(* Logix 5000 project; controller GEA_Test_Chamber vendor 1 type 14 code 196 rev 32.14; software revision 32.04; part 2 of 11 *)
(* tags used below, declared in another part *)
   Ref_Transactions : raC_UDT_ModbusClientTransaction[5];
   Sts_Overlap : BOOL;
   Sts_Overload : BOOL;
   Wrk_Main_Read_Buffer : STR4096;
   Wrk_ArraySize : DINT;
   Wrk_LastTransaction : DINT;
   Wrk_tempHMItransaction : DINT;
   Wrk_HMITransactionValid : BOOL;
(* raC_Opr_NetModbusTCPClient, continued *)

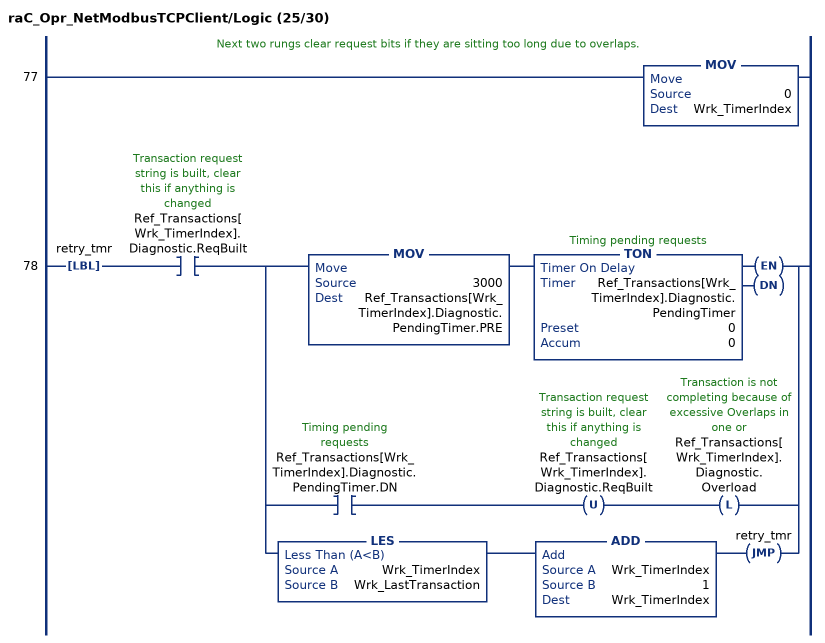
   // Next two rungs clear request bits if they are sitting too long due to overlaps.
   77: MOV(0,Wrk_TimerIndex);
   78: LBL(retry_tmr)XIC(Ref_Transactions[Wrk_TimerIndex].Diagnostic.ReqBuilt)[MOV(3000,Ref_Transactions[Wrk_TimerIndex].Diagnostic.PendingTimer.PRE) TON(Ref_Transactions[Wrk_TimerIndex].Diagnostic.PendingTimer,0,0) ,XIC(Ref_Transactions[Wrk_TimerIndex].Diagnostic.PendingTimer.DN) OTU(Ref_Transactions[Wrk_TimerIndex].Diagnostic.ReqBuilt) OTL(Ref_Transactions[Wrk_TimerIndex].Diagnostic.Overload) ,LES(Wrk_TimerIndex,Wrk_LastTransaction) ADD(Wrk_TimerIndex,1,Wrk_TimerIndex) JMP(retry_tmr) ];
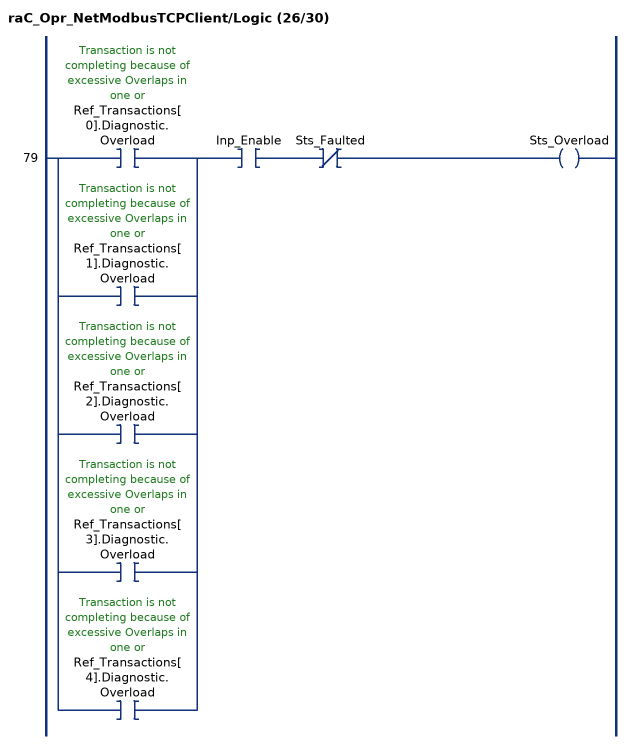
   79: [XIC(Ref_Transactions[0].Diagnostic.Overload) ,XIC(Ref_Transactions[1].Diagnostic.Overload) ,XIC(Ref_Transactions[2].Diagnostic.Overload) ,XIC(Ref_Transactions[3].Diagnostic.Overload) ,XIC(Ref_Transactions[4].Diagnostic.Overload) ]XIC(Inp_Enable)XIO(Sts_Faulted)OTE(Sts_Overload);
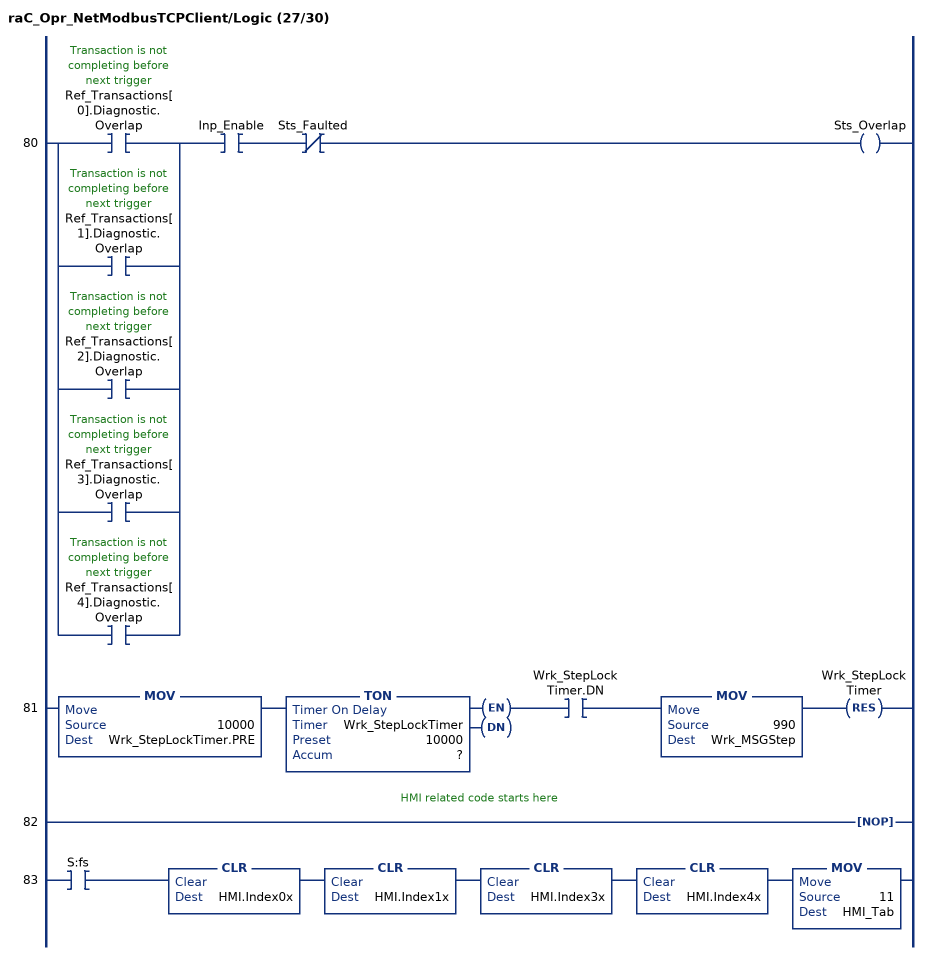
   80: [XIC(Ref_Transactions[0].Diagnostic.Overlap) ,XIC(Ref_Transactions[1].Diagnostic.Overlap) ,XIC(Ref_Transactions[2].Diagnostic.Overlap) ,XIC(Ref_Transactions[3].Diagnostic.Overlap) ,XIC(Ref_Transactions[4].Diagnostic.Overlap) ]XIC(Inp_Enable)XIO(Sts_Faulted)OTE(Sts_Overlap);
   81: MOV(10000,Wrk_StepLockTimer.PRE)TON(Wrk_StepLockTimer,?,?)XIC(Wrk_StepLockTimer.DN)MOV(990,Wrk_MSGStep)RES(Wrk_StepLockTimer);
   // HMI related code starts here
   82: NOP();
   83: XIC(S:fs)CLR(HMI.Index0x)CLR(HMI.Index1x)CLR(HMI.Index3x)CLR(HMI.Index4x)MOV(11,HMI_Tab);
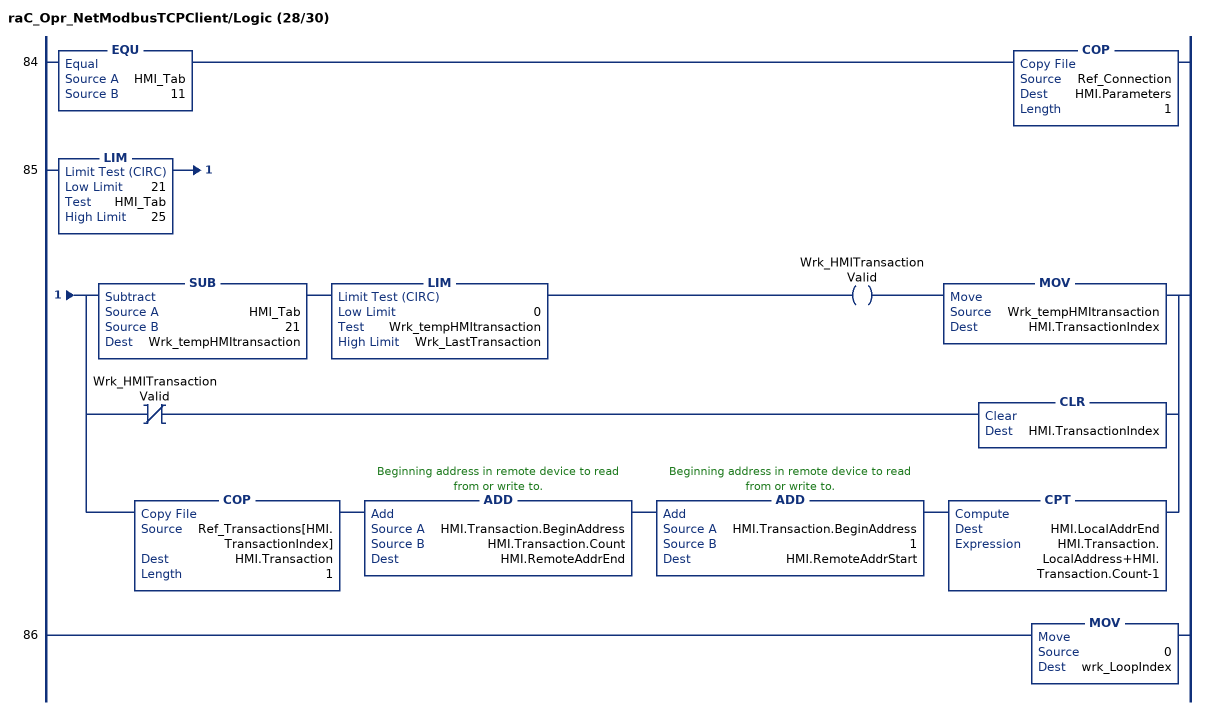
   84: EQU(HMI_Tab,11)COP(Ref_Connection,HMI.Parameters,1);
   85: LIM(21,HMI_Tab,25)[SUB(HMI_Tab,21,Wrk_tempHMItransaction) LIM(0,Wrk_tempHMItransaction,Wrk_LastTransaction) OTE(Wrk_HMITransactionValid) MOV(Wrk_tempHMItransaction,HMI.TransactionIndex) ,XIO(Wrk_HMITransactionValid) CLR(HMI.TransactionIndex) ,COP(Ref_Transactions[HMI.TransactionIndex],HMI.Transaction,1) ADD(HMI.Transaction.BeginAddress,HMI.Transaction.Count,HMI.RemoteAddrEnd) ADD(HMI.Transaction.BeginAddress,1,HMI.RemoteAddrStart) CPT(HMI.LocalAddrEnd,HMI.Transaction.LocalAddress+HMI.Transaction.Count-1) ];
   86: MOV(0,wrk_LoopIndex);
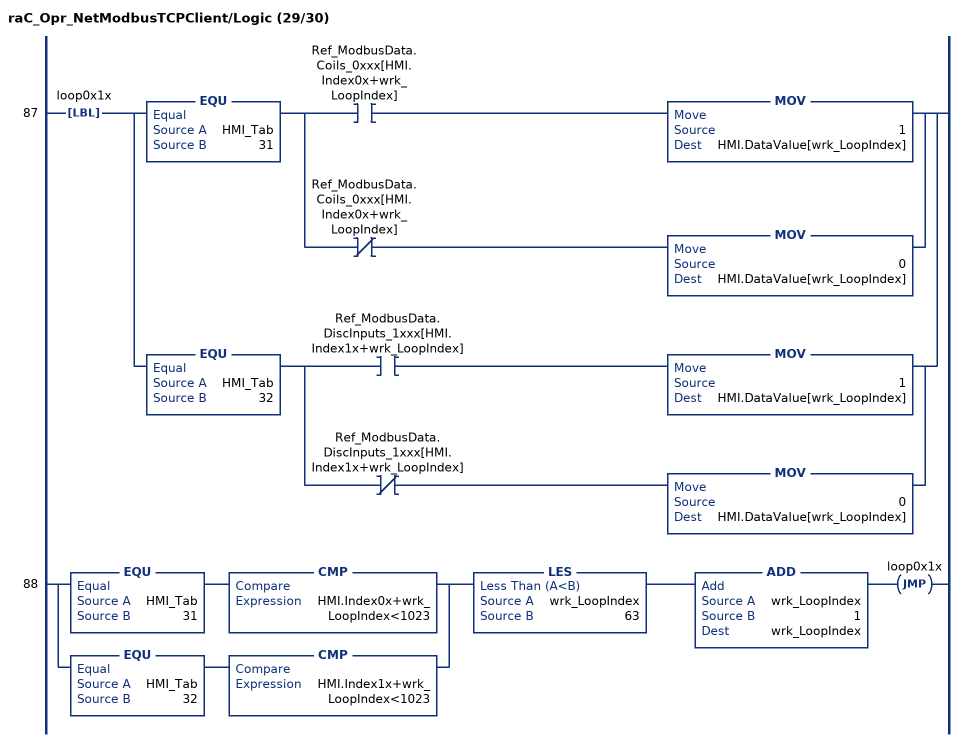
   87: LBL(loop0x1x)[EQU(HMI_Tab,31) [XIC(Ref_ModbusData.Coils_0xxx[HMI.Index0x+wrk_LoopIndex]) MOV(1,HMI.DataValue[wrk_LoopIndex]) ,XIO(Ref_ModbusData.Coils_0xxx[HMI.Index0x+wrk_LoopIndex]) MOV(0,HMI.DataValue[wrk_LoopIndex]) ] ,EQU(HMI_Tab,32) [XIC(Ref_ModbusData.DiscInputs_1xxx[HMI.Index1x+wrk_LoopIndex]) MOV(1,HMI.DataValue[wrk_LoopIndex]) ,XIO(Ref_ModbusData.DiscInputs_1xxx[HMI.Index1x+wrk_LoopIndex]) MOV(0,HMI.DataValue[wrk_LoopIndex]) ] ];
   88: [EQU(HMI_Tab,31) CMP(HMI.Index0x+wrk_LoopIndex<1023) ,EQU(HMI_Tab,32) CMP(HMI.Index1x+wrk_LoopIndex<1023) ]LES(wrk_LoopIndex,63)ADD(wrk_LoopIndex,1,wrk_LoopIndex)JMP(loop0x1x);
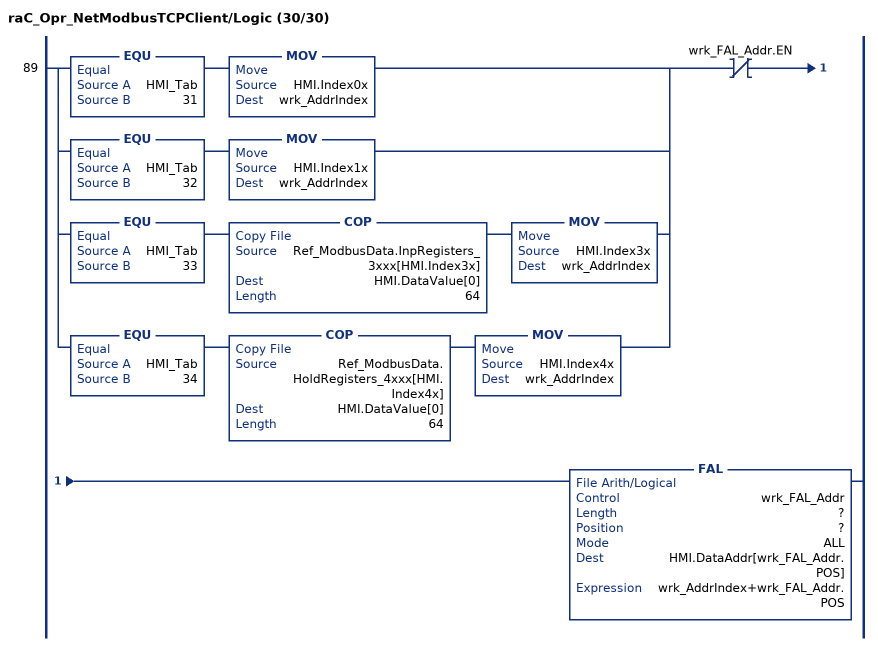
   89: [EQU(HMI_Tab,31) MOV(HMI.Index0x,wrk_AddrIndex) ,EQU(HMI_Tab,32) MOV(HMI.Index1x,wrk_AddrIndex) ,EQU(HMI_Tab,33) COP(Ref_ModbusData.InpRegisters_3xxx[HMI.Index3x],HMI.DataValue[0],64) MOV(HMI.Index3x,wrk_AddrIndex) ,EQU(HMI_Tab,34) COP(Ref_ModbusData.HoldRegisters_4xxx[HMI.Index4x],HMI.DataValue[0],64) MOV(HMI.Index4x,wrk_AddrIndex) ]XIO(wrk_FAL_Addr.EN)FAL(wrk_FAL_Addr,?,?,ALL,HMI.DataAddr[wrk_FAL_Addr.POS],wrk_AddrIndex+wrk_FAL_Addr.POS);
END_ROUTINE

ROUTINE Prescan   (* ladder *)
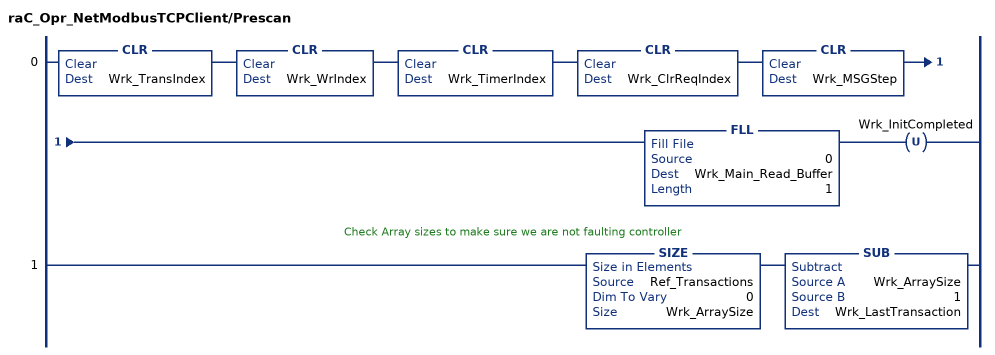
   0: CLR(Wrk_TransIndex)CLR(Wrk_WrIndex)CLR(Wrk_TimerIndex)CLR(Wrk_ClrReqIndex)CLR(Wrk_MSGStep)FLL(0,Wrk_Main_Read_Buffer,1)OTU(Wrk_InitCompleted);
   // Check Array sizes to make sure we are not faulting controller
   1: SIZE(Ref_Transactions,0,Wrk_ArraySize)SUB(Wrk_ArraySize,1,Wrk_LastTransaction);
END_ROUTINE
END_ADD_ON_INSTRUCTION

ADD_ON_INSTRUCTION raC_Opr_NetModbusTCPServer   (* revision 2.3 0, vendor Rockwell Automation, ExecutePrescan *)
// Modbus TCP Server
// Revision note:
// 2.0.0 Initial release in AOI format
// 2.0.1 Corrected local IP address logic
// 2.1.0 Corrected power-up and Redundancy anomalies
// 2.2.0 Force LocalSlot 0 for CompactLogix
// 2.3.0 Added incoming Client IP address reference tag and HMI structure
VAR_INPUT
   Inp_Enable : BOOL; {required}
END_VAR
VAR_IN_OUT
   Ref_Connection : raC_UDT_ModbusServerBase; {required}
   Ref_ModbusData : raC_UDT_ModbusServerData; {required}
END_VAR
VAR_OUTPUT
   Sts_ActiveConnections : DINT; {access Read Only, visible}   // Number of currently active Client connections.
END_VAR
VAR_IN_OUT
   Ref_MsgCreate : MESSAGE; {required}
   Ref_MsgAccept : MESSAGE; {required}
   Ref_MsgRead : MESSAGE; {required}
   Ref_MsgWrite : MESSAGE; {required}
   Ref_MsgDelete : MESSAGE; {required}
   Ref_MsgDeleteAll : MESSAGE; {required}
   Ref_MsgSetAttrSingle : MESSAGE; {required}
END_VAR
VAR_OUTPUT
   Sts_EN : BOOL; {access Read Only, visible}
   Sts_Waiting : BOOL; {access Read Only, visible}
   Sts_Accepted : BOOL; {access Read Only, visible}
   Sts_Faulted : BOOL; {access Read Only, visible}
   Sts_LastError : DINT; {access Read Only}   // The last recorded socket error for this connection. 0 good, -2- Write Error, -4 - Read Error, -6 connection failed, -7 Delete all failed, -8 Create Soc failed, -9 Connection failed, -10 connection dropped, -11 error in setting socket parameter. -12 - Enable removed -15 - Max number of connected clients exceeded
END_VAR
VAR
   Wrk_MSGStep : DINT; {access None}
   Wrk_CreateReq : raC_UDT_ModbusCreateParam; {access None}
   Wrk_BaseInstance : DINT; {access None}
   Wrk_NoreplyCounter : DINT; {access None}
   Wrk_RetryTimer : TIMER := (PRE := 5000); {access None}
   Wrk_MSGRead_SRC : DINT[2]; {access None}   // User for MSG Read Source
   Wrk_TempString : STR0462; {access None}
   Wrk_WrIndex : DINT; {access None}
   Wrk_TempDINT : DINT; {access None}
   Wrk_AdditionalLen : INT; {access None}
   Wrk_AdditionaLenRead : INT; {access None}
   Wrk_ModbusCmdLen : INT; {access None}
   Wrk_AdditionalLen1 : INT; {access None}
   Wrk_ModbusPacket : STR0462; {access None}
   Wrk_DataReceived : BOOL; {access None}
   Wrk_CmdFromReadPacket : DINT; {access None}
   Wrk_ModbusID : STR0008; {access None}
   Wrk_TempInt : INT; {access None}
   Wrk_ModbusCmdStart : INT; {access None}
   Wrk_ModbusUnit : STR0008; {access None}
   Wrk_ModbusBytes : DINT; {access None}
   Wrk_ModbusCmdString : STR0462; {access None}
   Wrk_RSB : raC_Tec_NetModbusTCPServer_RespStrBit; {access None}
   Wrk_TransIndex : DINT; {access None}
   Wrk_TimerIndex : DINT; {access None}
   Wrk_RSW : raC_Tec_NetModbusTCPServer_RespStrWord; {access None}
   Wrk_TempOctet : DINT[4]; {access None}
   Wrk_TempStrOctet : STR0008; {access None}
   Wrk_TempStrOctetlen : DINT; {access None}
   Wrk_TempIPStr : STR0016; {access None}
   Wrk_ClrReqIndex : DINT; {access None}
   Wrk_ListenSocketLost : BOOL; {access None}
   Wrk_AcceptInstance : DINT; {access None}
   Wrk_FES : raC_Tec_NetModbusTCPServer_FndEmptySckt; {access None}
   Wrk_InstSize : DINT; {access None}
   Wrk_RdWrIndex : DINT; {access None}
   Wrk_ModbusRespString : STR0462; {access None}
   Wrk_TempActConn : DINT; {access None}
   Wrk_InstIndex : DINT; {access None}
   Wrk_LastInstIndex : DINT; {access None}
   Wrk_OkToIncement : BOOL; {access None}
   Wrk_CmdFromReadPacketTmp : DINT; {access None}
   Wrk_StepLockTimer : TIMER := (PRE := 10000); {access None}
   Wrk_TempTime : DINT; {access None}
   Wrk_OktoCheckAccept : BOOL; {access None}
   Wrk_OkToIncement320 : BOOL; {access None}
   Wrk_Instances : raC_UDT_ModbusServerRWSocket[10]; {access Read Only}
   Wrk_Controller_Type : DINT; {access None}
   Wrk_Controller_Name : SINT[33]; {access None}
   Wrk_InitCompleted : BOOL; {access None}
   Wrk_AcceptAddress : DINT; {access None}
   Wrk_InstIndex2 : DINT; {access None}
   Wrk_InstIndex3 : DINT; {access None}
   HMI_Tab : DINT;
   Inf_Lib : STR0016; {access Read Only}
   Inf_Type : STR0032; {access Read Only}
   Inf_Version : STR0016; {access Read Only}
   wrk_temp_Instances : raC_UDT_ModbusServerRWSocketInfo[10]; {access None}
   wrk_FAL_Addr : CONTROL := (LEN := 64); {access None}
   wrk_LoopIndex : DINT; {access None}
   wrk_AddrIndex : DINT; {access None}
   HMI : raC_UDT_ModbusServerHMI;
   wrk_FAL_01 : CONTROL := (LEN := 10); {access None}
END_VAR

ROUTINE Logic   (* ladder *)
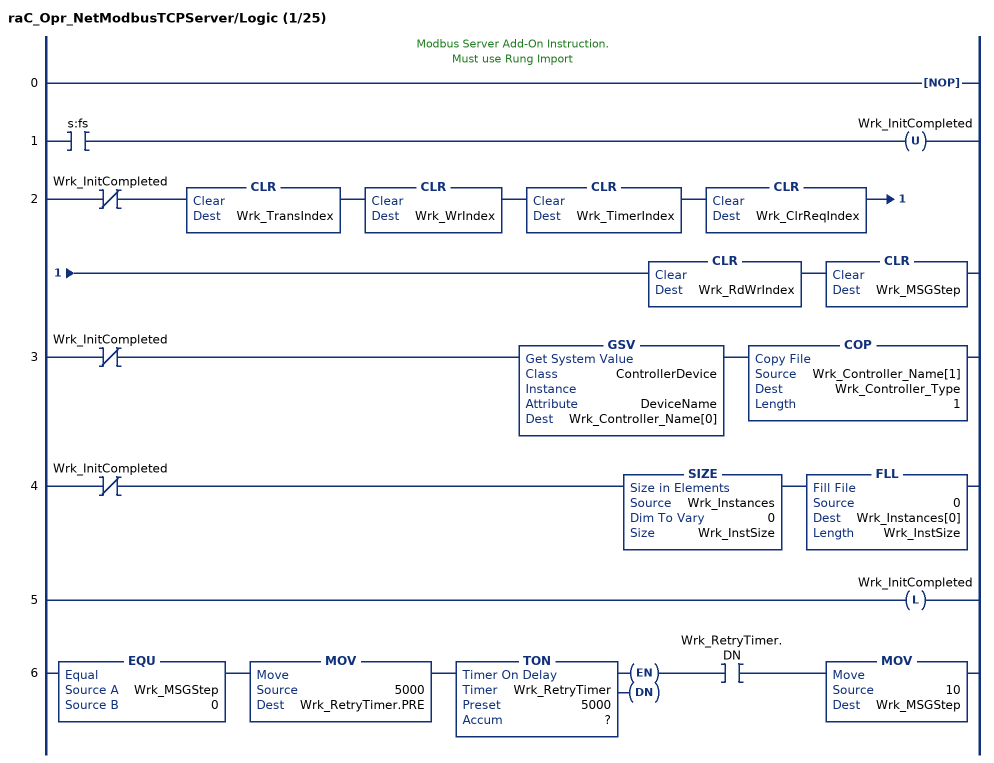
   // Modbus Server Add-On Instruction.
   // Must use Rung Import
   0: NOP();
   1: XIC(s:fs)OTU(Wrk_InitCompleted);
   2: XIO(Wrk_InitCompleted)CLR(Wrk_TransIndex)CLR(Wrk_WrIndex)CLR(Wrk_TimerIndex)CLR(Wrk_ClrReqIndex)CLR(Wrk_RdWrIndex)CLR(Wrk_MSGStep);
   3: XIO(Wrk_InitCompleted)GSV(ControllerDevice,,DeviceName,Wrk_Controller_Name[0])COP(Wrk_Controller_Name[1],Wrk_Controller_Type,1);
   4: XIO(Wrk_InitCompleted)SIZE(Wrk_Instances,0,Wrk_InstSize)FLL(0,Wrk_Instances[0],Wrk_InstSize);
   5: OTL(Wrk_InitCompleted);
   6: EQU(Wrk_MSGStep,0)MOV(5000,Wrk_RetryTimer.PRE)TON(Wrk_RetryTimer,?,?)XIC(Wrk_RetryTimer.DN)MOV(10,Wrk_MSGStep);
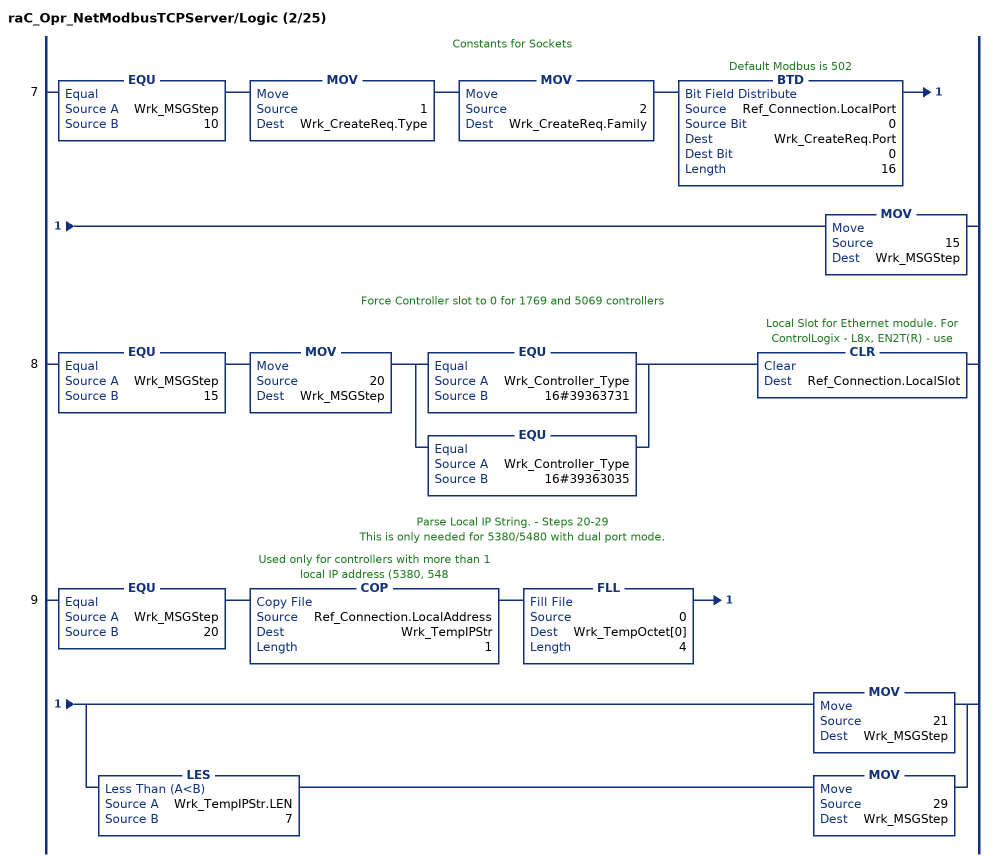
   // Constants for Sockets
   7: EQU(Wrk_MSGStep,10)MOV(1,Wrk_CreateReq.Type)MOV(2,Wrk_CreateReq.Family)BTD(Ref_Connection.LocalPort,0,Wrk_CreateReq.Port,0,16)MOV(15,Wrk_MSGStep);
   // Force Controller slot to 0 for 1769 and 5069 controllers
   8: EQU(Wrk_MSGStep,15)MOV(20,Wrk_MSGStep)[EQU(Wrk_Controller_Type,16#39363731) ,EQU(Wrk_Controller_Type,16#39363035) ]CLR(Ref_Connection.LocalSlot);
   // Parse Local IP String. - Steps 20-29
   // This is only needed for 5380/5480 with dual port mode.
   9: EQU(Wrk_MSGStep,20)COP(Ref_Connection.LocalAddress,Wrk_TempIPStr,1)FLL(0,Wrk_TempOctet[0],4)[MOV(21,Wrk_MSGStep) ,LES(Wrk_TempIPStr.LEN,7) MOV(29,Wrk_MSGStep) ];
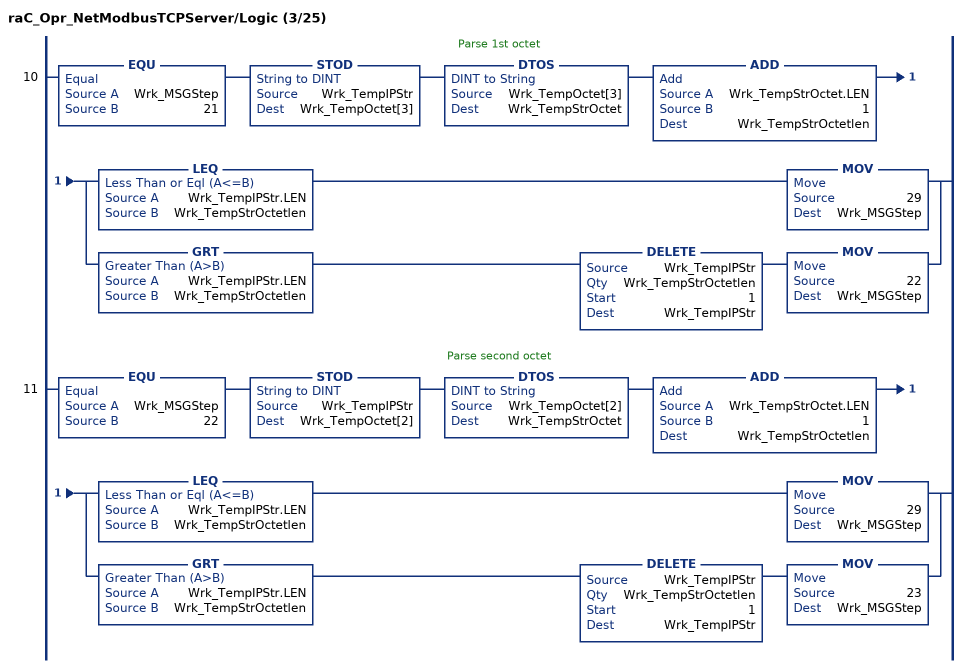
   // Parse 1st octet
   10: EQU(Wrk_MSGStep,21)STOD(Wrk_TempIPStr,Wrk_TempOctet[3])DTOS(Wrk_TempOctet[3],Wrk_TempStrOctet)ADD(Wrk_TempStrOctet.LEN,1,Wrk_TempStrOctetlen)[LEQ(Wrk_TempIPStr.LEN,Wrk_TempStrOctetlen) MOV(29,Wrk_MSGStep) ,GRT(Wrk_TempIPStr.LEN,Wrk_TempStrOctetlen) DELETE(Wrk_TempIPStr,Wrk_TempStrOctetlen,1,Wrk_TempIPStr) MOV(22,Wrk_MSGStep) ];
   // Parse second octet
   11: EQU(Wrk_MSGStep,22)STOD(Wrk_TempIPStr,Wrk_TempOctet[2])DTOS(Wrk_TempOctet[2],Wrk_TempStrOctet)ADD(Wrk_TempStrOctet.LEN,1,Wrk_TempStrOctetlen)[LEQ(Wrk_TempIPStr.LEN,Wrk_TempStrOctetlen) MOV(29,Wrk_MSGStep) ,GRT(Wrk_TempIPStr.LEN,Wrk_TempStrOctetlen) DELETE(Wrk_TempIPStr,Wrk_TempStrOctetlen,1,Wrk_TempIPStr) MOV(23,Wrk_MSGStep) ];
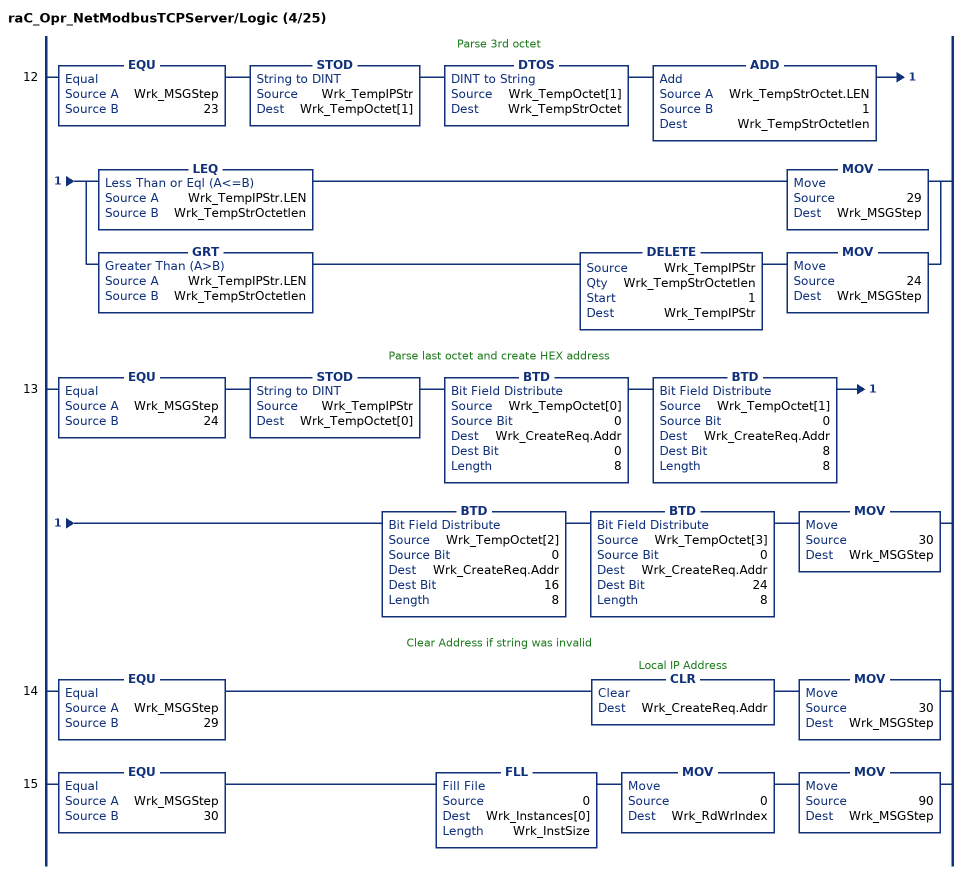
   // Parse 3rd octet
   12: EQU(Wrk_MSGStep,23)STOD(Wrk_TempIPStr,Wrk_TempOctet[1])DTOS(Wrk_TempOctet[1],Wrk_TempStrOctet)ADD(Wrk_TempStrOctet.LEN,1,Wrk_TempStrOctetlen)[LEQ(Wrk_TempIPStr.LEN,Wrk_TempStrOctetlen) MOV(29,Wrk_MSGStep) ,GRT(Wrk_TempIPStr.LEN,Wrk_TempStrOctetlen) DELETE(Wrk_TempIPStr,Wrk_TempStrOctetlen,1,Wrk_TempIPStr) MOV(24,Wrk_MSGStep) ];
   // Parse last octet and create HEX address
   13: EQU(Wrk_MSGStep,24)STOD(Wrk_TempIPStr,Wrk_TempOctet[0])BTD(Wrk_TempOctet[0],0,Wrk_CreateReq.Addr,0,8)BTD(Wrk_TempOctet[1],0,Wrk_CreateReq.Addr,8,8)BTD(Wrk_TempOctet[2],0,Wrk_CreateReq.Addr,16,8)BTD(Wrk_TempOctet[3],0,Wrk_CreateReq.Addr,24,8)MOV(30,Wrk_MSGStep);
   // Clear Address if string was invalid
   14: EQU(Wrk_MSGStep,29)CLR(Wrk_CreateReq.Addr)MOV(30,Wrk_MSGStep);
   15: EQU(Wrk_MSGStep,30)FLL(0,Wrk_Instances[0],Wrk_InstSize)MOV(0,Wrk_RdWrIndex)MOV(90,Wrk_MSGStep);
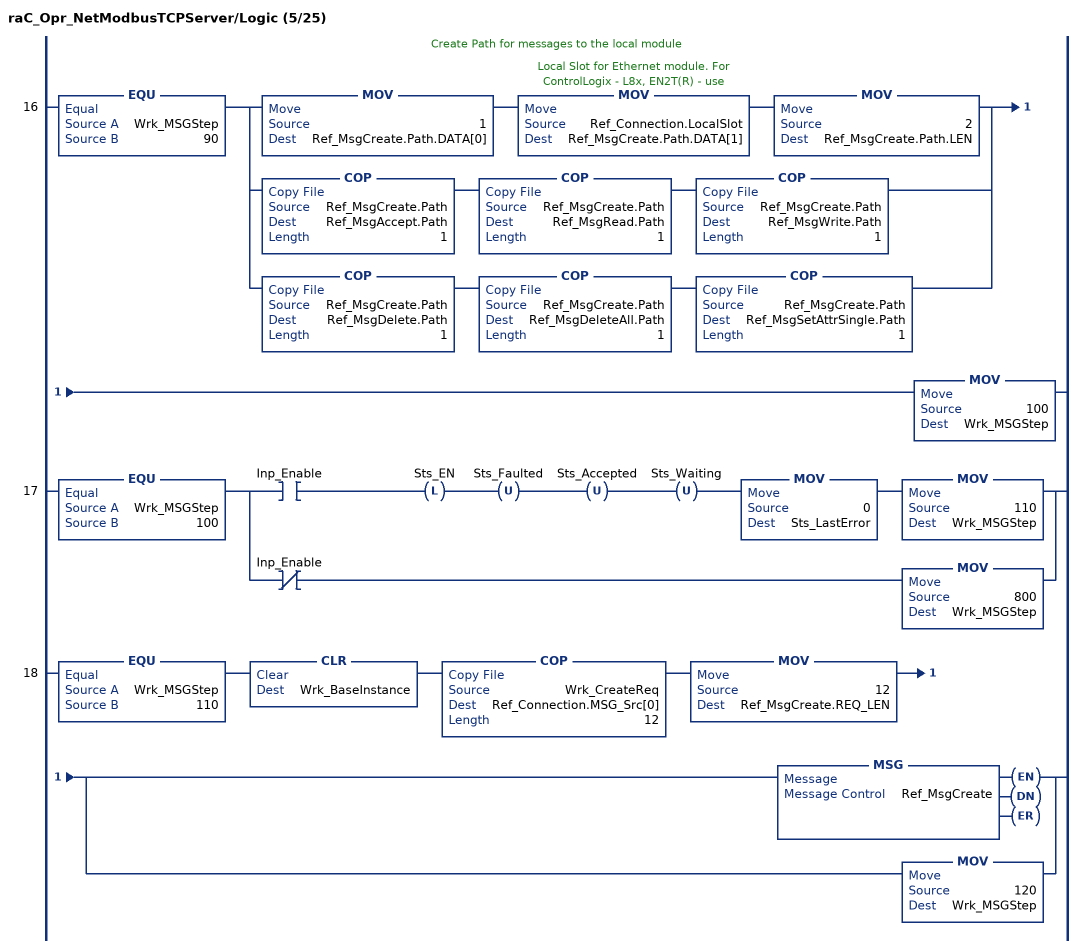
   // Create Path for messages to the local module
   16: EQU(Wrk_MSGStep,90)[MOV(1,Ref_MsgCreate.Path.DATA[0]) MOV(Ref_Connection.LocalSlot,Ref_MsgCreate.Path.DATA[1]) MOV(2,Ref_MsgCreate.Path.LEN) ,COP(Ref_MsgCreate.Path,Ref_MsgAccept.Path,1) COP(Ref_MsgCreate.Path,Ref_MsgRead.Path,1) COP(Ref_MsgCreate.Path,Ref_MsgWrite.Path,1) ,COP(Ref_MsgCreate.Path,Ref_MsgDelete.Path,1) COP(Ref_MsgCreate.Path,Ref_MsgDeleteAll.Path,1) COP(Ref_MsgCreate.Path,Ref_MsgSetAttrSingle.Path,1) ]MOV(100,Wrk_MSGStep);
   17: EQU(Wrk_MSGStep,100)[XIC(Inp_Enable) OTL(Sts_EN) OTU(Sts_Faulted) OTU(Sts_Accepted) OTU(Sts_Waiting) MOV(0,Sts_LastError) MOV(110,Wrk_MSGStep) ,XIO(Inp_Enable) MOV(800,Wrk_MSGStep) ];
   18: EQU(Wrk_MSGStep,110)CLR(Wrk_BaseInstance)COP(Wrk_CreateReq,Ref_Connection.MSG_Src[0],12)MOV(12,Ref_MsgCreate.REQ_LEN)[MSG(Ref_MsgCreate) ,MOV(120,Wrk_MSGStep) ];
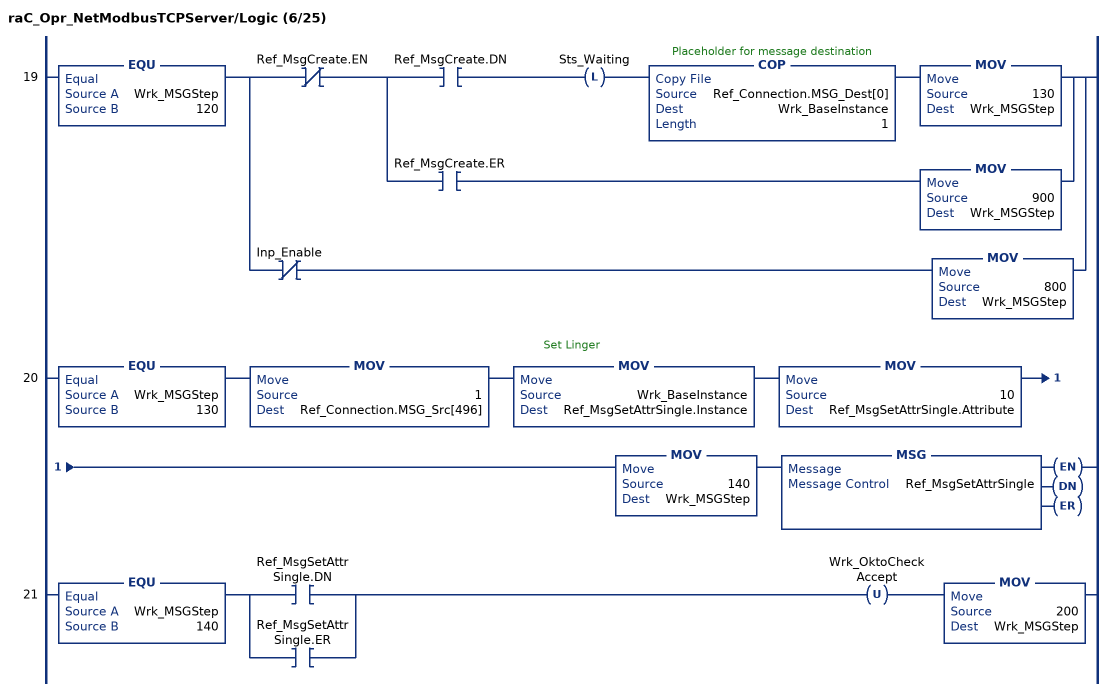
   19: EQU(Wrk_MSGStep,120)[XIO(Ref_MsgCreate.EN) [XIC(Ref_MsgCreate.DN) OTL(Sts_Waiting) COP(Ref_Connection.MSG_Dest[0],Wrk_BaseInstance,1) MOV(130,Wrk_MSGStep) ,XIC(Ref_MsgCreate.ER) MOV(900,Wrk_MSGStep) ] ,XIO(Inp_Enable) MOV(800,Wrk_MSGStep) ];
   // Set Linger
   20: EQU(Wrk_MSGStep,130)MOV(1,Ref_Connection.MSG_Src[496])MOV(Wrk_BaseInstance,Ref_MsgSetAttrSingle.Instance)MOV(10,Ref_MsgSetAttrSingle.Attribute)MOV(140,Wrk_MSGStep)MSG(Ref_MsgSetAttrSingle);
   21: EQU(Wrk_MSGStep,140)[XIC(Ref_MsgSetAttrSingle.DN) ,XIC(Ref_MsgSetAttrSingle.ER) ]OTU(Wrk_OktoCheckAccept)MOV(200,Wrk_MSGStep);
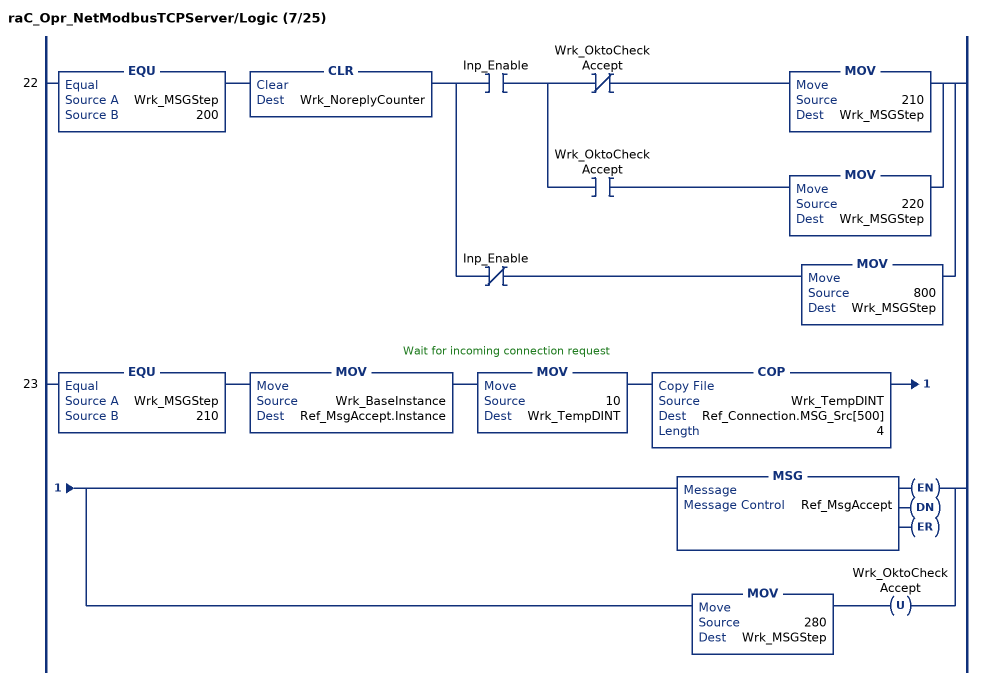
   22: EQU(Wrk_MSGStep,200)CLR(Wrk_NoreplyCounter)[XIC(Inp_Enable) [XIO(Wrk_OktoCheckAccept) MOV(210,Wrk_MSGStep) ,XIC(Wrk_OktoCheckAccept) MOV(220,Wrk_MSGStep) ] ,XIO(Inp_Enable) MOV(800,Wrk_MSGStep) ];
   // Wait for incoming connection request
   23: EQU(Wrk_MSGStep,210)MOV(Wrk_BaseInstance,Ref_MsgAccept.Instance)MOV(10,Wrk_TempDINT)COP(Wrk_TempDINT,Ref_Connection.MSG_Src[500],4)[MSG(Ref_MsgAccept) ,MOV(280,Wrk_MSGStep) OTU(Wrk_OktoCheckAccept) ];
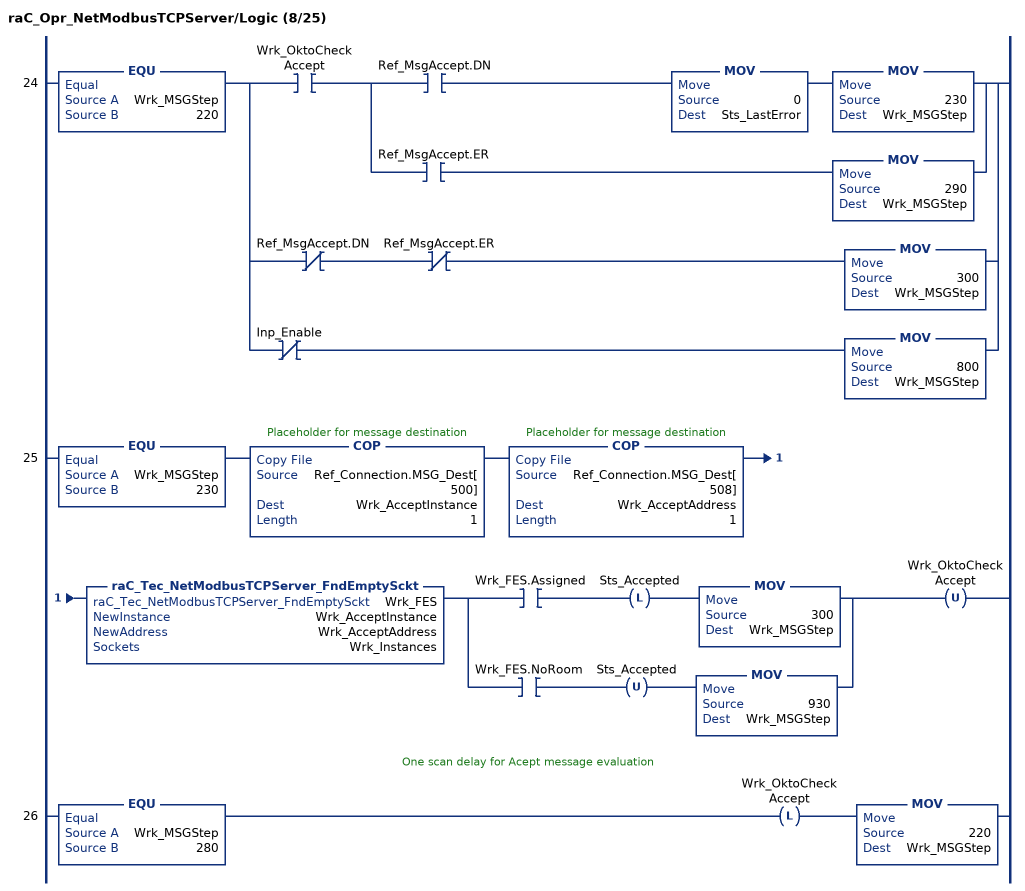
   24: EQU(Wrk_MSGStep,220)[XIC(Wrk_OktoCheckAccept) [XIC(Ref_MsgAccept.DN) MOV(0,Sts_LastError) MOV(230,Wrk_MSGStep) ,XIC(Ref_MsgAccept.ER) MOV(290,Wrk_MSGStep) ] ,XIO(Ref_MsgAccept.DN) XIO(Ref_MsgAccept.ER) MOV(300,Wrk_MSGStep) ,XIO(Inp_Enable) MOV(800,Wrk_MSGStep) ];
   25: EQU(Wrk_MSGStep,230)COP(Ref_Connection.MSG_Dest[500],Wrk_AcceptInstance,1)COP(Ref_Connection.MSG_Dest[508],Wrk_AcceptAddress,1)raC_Tec_NetModbusTCPServer_FndEmptySckt(Wrk_FES,Wrk_AcceptInstance,Wrk_AcceptAddress,Wrk_Instances)[XIC(Wrk_FES.Assigned) OTL(Sts_Accepted) MOV(300,Wrk_MSGStep) ,XIC(Wrk_FES.NoRoom) OTU(Sts_Accepted) MOV(930,Wrk_MSGStep) ]OTU(Wrk_OktoCheckAccept);
   // One scan delay for Acept message evaluation
   26: EQU(Wrk_MSGStep,280)OTL(Wrk_OktoCheckAccept)MOV(220,Wrk_MSGStep);
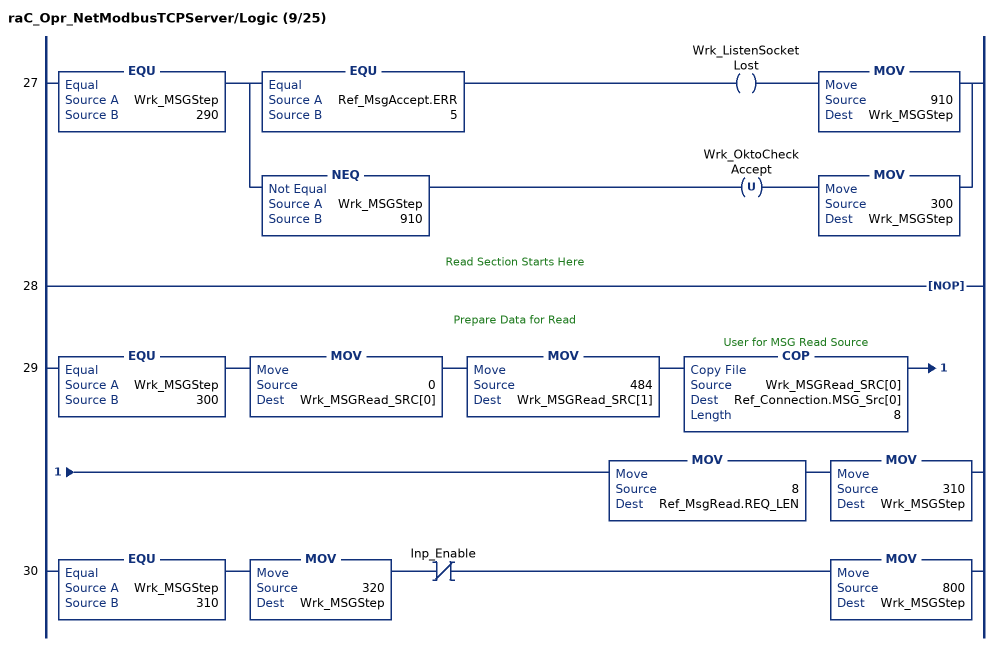
   27: EQU(Wrk_MSGStep,290)[EQU(Ref_MsgAccept.ERR,5) OTE(Wrk_ListenSocketLost) MOV(910,Wrk_MSGStep) ,NEQ(Wrk_MSGStep,910) OTU(Wrk_OktoCheckAccept) MOV(300,Wrk_MSGStep) ];
   // Read Section Starts Here
   28: NOP();
   // Prepare Data for Read
   29: EQU(Wrk_MSGStep,300)MOV(0,Wrk_MSGRead_SRC[0])MOV(484,Wrk_MSGRead_SRC[1])COP(Wrk_MSGRead_SRC[0],Ref_Connection.MSG_Src[0],8)MOV(8,Ref_MsgRead.REQ_LEN)MOV(310,Wrk_MSGStep);
   30: EQU(Wrk_MSGStep,310)MOV(320,Wrk_MSGStep)XIO(Inp_Enable)MOV(800,Wrk_MSGStep);
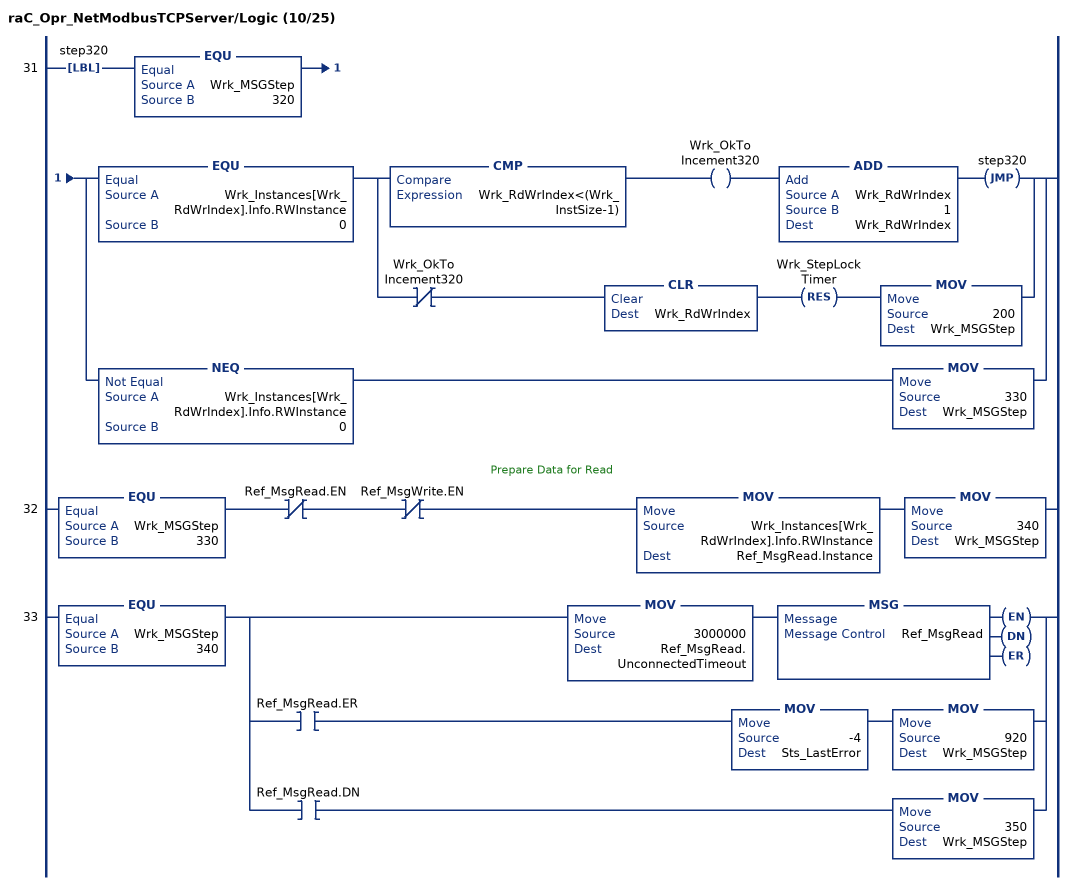
   31: LBL(step320)EQU(Wrk_MSGStep,320)[EQU(Wrk_Instances[Wrk_RdWrIndex].Info.RWInstance,0) [CMP(Wrk_RdWrIndex<(Wrk_InstSize-1)) OTE(Wrk_OkToIncement320) ADD(Wrk_RdWrIndex,1,Wrk_RdWrIndex) JMP(step320) ,XIO(Wrk_OkToIncement320) CLR(Wrk_RdWrIndex) RES(Wrk_StepLockTimer) MOV(200,Wrk_MSGStep) ] ,NEQ(Wrk_Instances[Wrk_RdWrIndex].Info.RWInstance,0) MOV(330,Wrk_MSGStep) ];
   // Prepare Data for Read
   32: EQU(Wrk_MSGStep,330)XIO(Ref_MsgRead.EN)XIO(Ref_MsgWrite.EN)MOV(Wrk_Instances[Wrk_RdWrIndex].Info.RWInstance,Ref_MsgRead.Instance)MOV(340,Wrk_MSGStep);
   33: EQU(Wrk_MSGStep,340)[MOV(3000000,Ref_MsgRead.UnconnectedTimeout) MSG(Ref_MsgRead) ,XIC(Ref_MsgRead.ER) MOV(-4,Sts_LastError) MOV(920,Wrk_MSGStep) ,XIC(Ref_MsgRead.DN) MOV(350,Wrk_MSGStep) ];
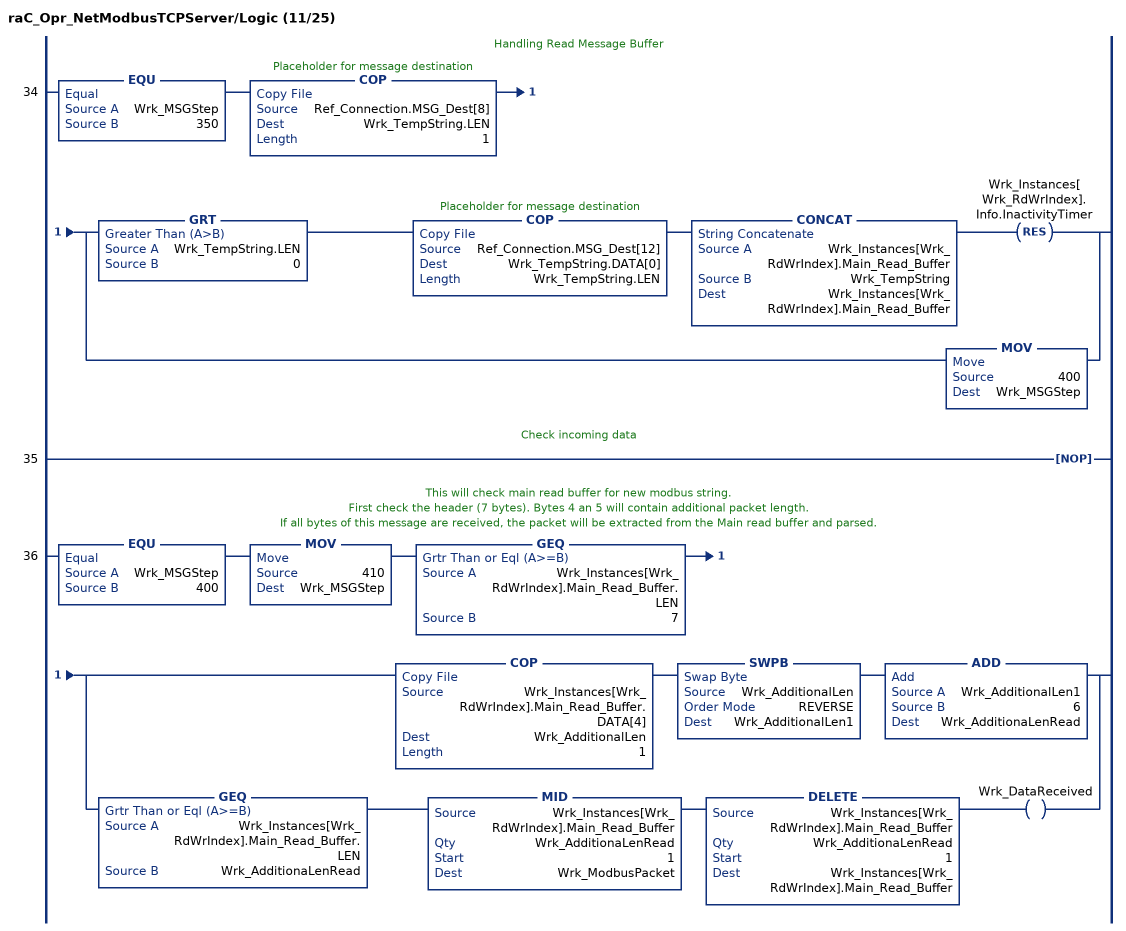
   // Handling Read Message Buffer
   34: EQU(Wrk_MSGStep,350)COP(Ref_Connection.MSG_Dest[8],Wrk_TempString.LEN,1)[GRT(Wrk_TempString.LEN,0) COP(Ref_Connection.MSG_Dest[12],Wrk_TempString.DATA[0],Wrk_TempString.LEN) CONCAT(Wrk_Instances[Wrk_RdWrIndex].Main_Read_Buffer,Wrk_TempString,Wrk_Instances[Wrk_RdWrIndex].Main_Read_Buffer) RES(Wrk_Instances[Wrk_RdWrIndex].Info.InactivityTimer) ,MOV(400,Wrk_MSGStep) ];
   // Check incoming data
   35: NOP();
   // This will check main read buffer for new modbus string.
   // First check the header (7 bytes). Bytes 4 an 5 will contain additional packet length.
   // If all bytes of this message are received, the packet will be extracted from the Main read buffer and parsed.
   36: EQU(Wrk_MSGStep,400)MOV(410,Wrk_MSGStep)GEQ(Wrk_Instances[Wrk_RdWrIndex].Main_Read_Buffer.LEN,7)[COP(Wrk_Instances[Wrk_RdWrIndex].Main_Read_Buffer.DATA[4],Wrk_AdditionalLen,1) SWPB(Wrk_AdditionalLen,REVERSE,Wrk_AdditionalLen1) ADD(Wrk_AdditionalLen1,6,Wrk_AdditionaLenRead) ,GEQ(Wrk_Instances[Wrk_RdWrIndex].Main_Read_Buffer.LEN,Wrk_AdditionaLenRead) MID(Wrk_Instances[Wrk_RdWrIndex].Main_Read_Buffer,Wrk_AdditionaLenRead,1,Wrk_ModbusPacket) DELETE(Wrk_Instances[Wrk_RdWrIndex].Main_Read_Buffer,Wrk_AdditionaLenRead,1,Wrk_Instances[Wrk_RdWrIndex].Main_Read_Buffer) OTE(Wrk_DataReceived) ];
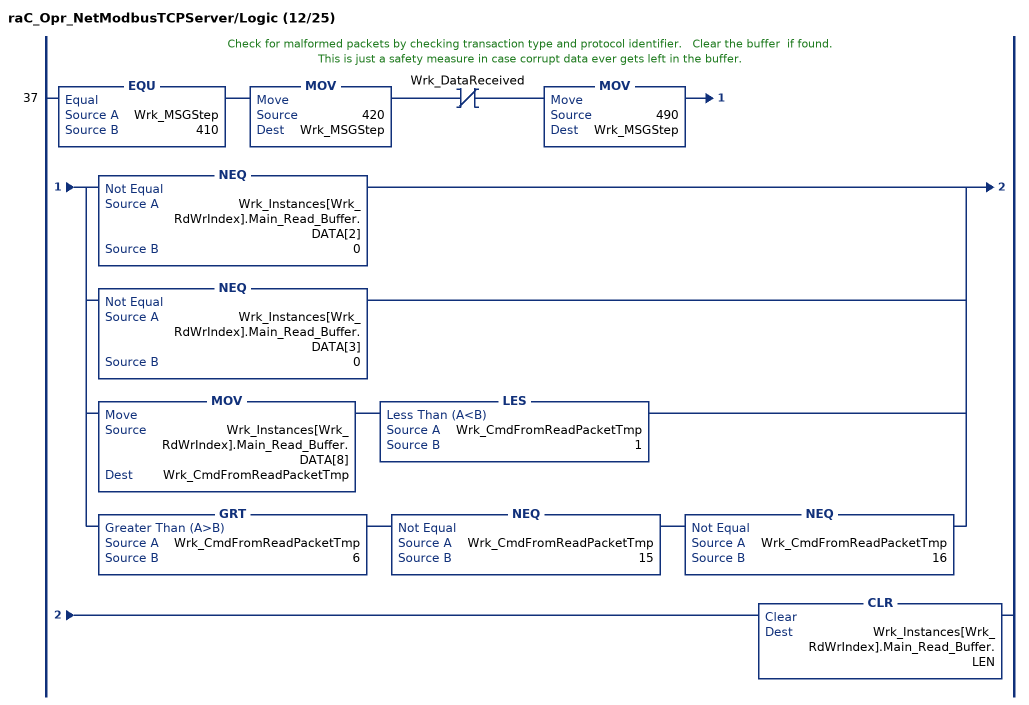
   // Check for malformed packets by checking transaction type and protocol identifier.   Clear the buffer  if found.
   // This is just a safety measure in case corrupt data ever gets left in the buffer.
   37: EQU(Wrk_MSGStep,410)MOV(420,Wrk_MSGStep)XIO(Wrk_DataReceived)MOV(490,Wrk_MSGStep)[NEQ(Wrk_Instances[Wrk_RdWrIndex].Main_Read_Buffer.DATA[2],0) ,NEQ(Wrk_Instances[Wrk_RdWrIndex].Main_Read_Buffer.DATA[3],0) ,MOV(Wrk_Instances[Wrk_RdWrIndex].Main_Read_Buffer.DATA[8],Wrk_CmdFromReadPacketTmp) LES(Wrk_CmdFromReadPacketTmp,1) ,GRT(Wrk_CmdFromReadPacketTmp,6) NEQ(Wrk_CmdFromReadPacketTmp,15) NEQ(Wrk_CmdFromReadPacketTmp,16) ]CLR(Wrk_Instances[Wrk_RdWrIndex].Main_Read_Buffer.LEN);
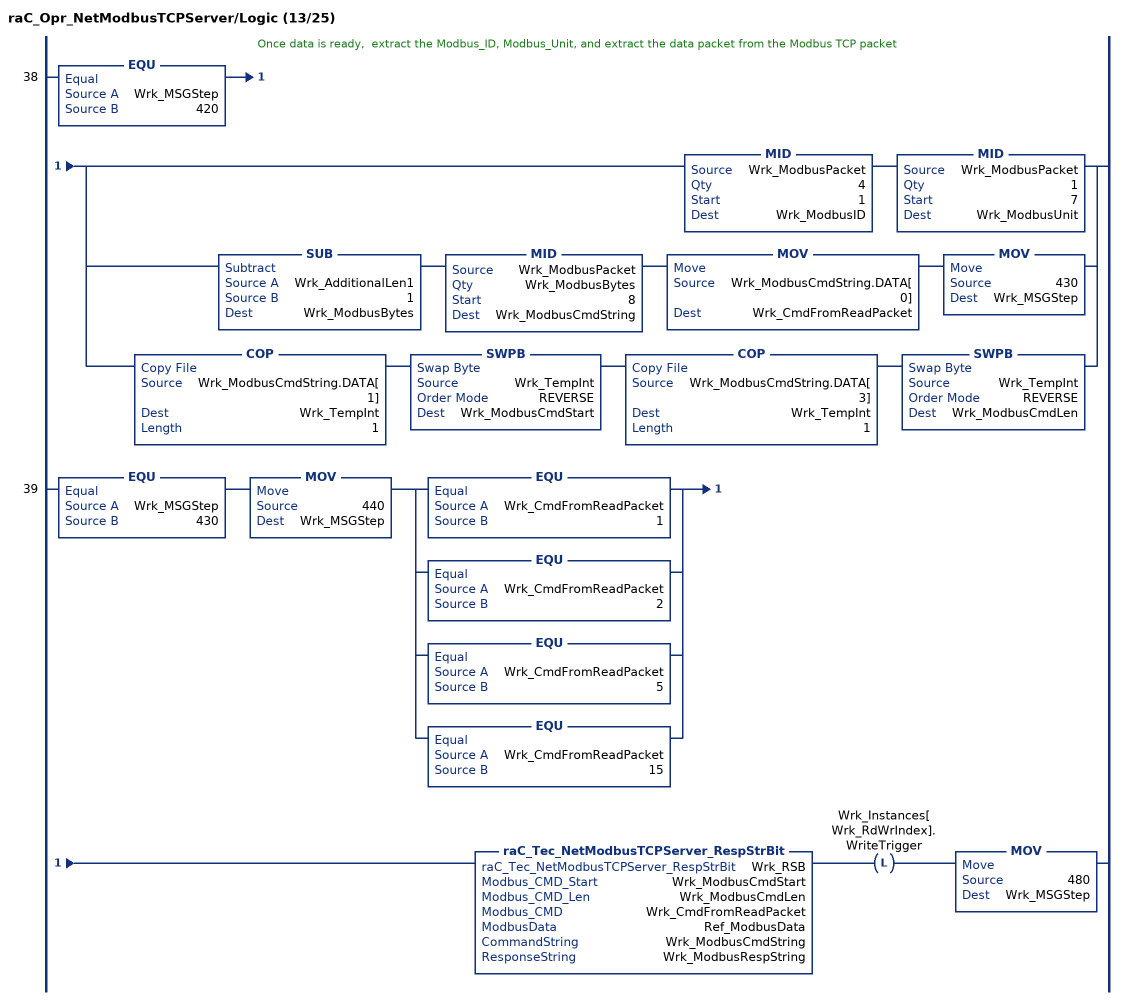
   // Once data is ready,  extract the Modbus_ID, Modbus_Unit, and extract the data packet from the Modbus TCP packet
   38: EQU(Wrk_MSGStep,420)[MID(Wrk_ModbusPacket,4,1,Wrk_ModbusID) MID(Wrk_ModbusPacket,1,7,Wrk_ModbusUnit) ,SUB(Wrk_AdditionalLen1,1,Wrk_ModbusBytes) MID(Wrk_ModbusPacket,Wrk_ModbusBytes,8,Wrk_ModbusCmdString) MOV(Wrk_ModbusCmdString.DATA[0],Wrk_CmdFromReadPacket) MOV(430,Wrk_MSGStep) ,COP(Wrk_ModbusCmdString.DATA[1],Wrk_TempInt,1) SWPB(Wrk_TempInt,REVERSE,Wrk_ModbusCmdStart) COP(Wrk_ModbusCmdString.DATA[3],Wrk_TempInt,1) SWPB(Wrk_TempInt,REVERSE,Wrk_ModbusCmdLen) ];
   39: EQU(Wrk_MSGStep,430)MOV(440,Wrk_MSGStep)[EQU(Wrk_CmdFromReadPacket,1) ,EQU(Wrk_CmdFromReadPacket,2) ,EQU(Wrk_CmdFromReadPacket,5) ,EQU(Wrk_CmdFromReadPacket,15) ]raC_Tec_NetModbusTCPServer_RespStrBit(Wrk_RSB,Wrk_ModbusCmdStart,Wrk_ModbusCmdLen,Wrk_CmdFromReadPacket,Ref_ModbusData,Wrk_ModbusCmdString,Wrk_ModbusRespString)OTL(Wrk_Instances[Wrk_RdWrIndex].WriteTrigger)MOV(480,Wrk_MSGStep);
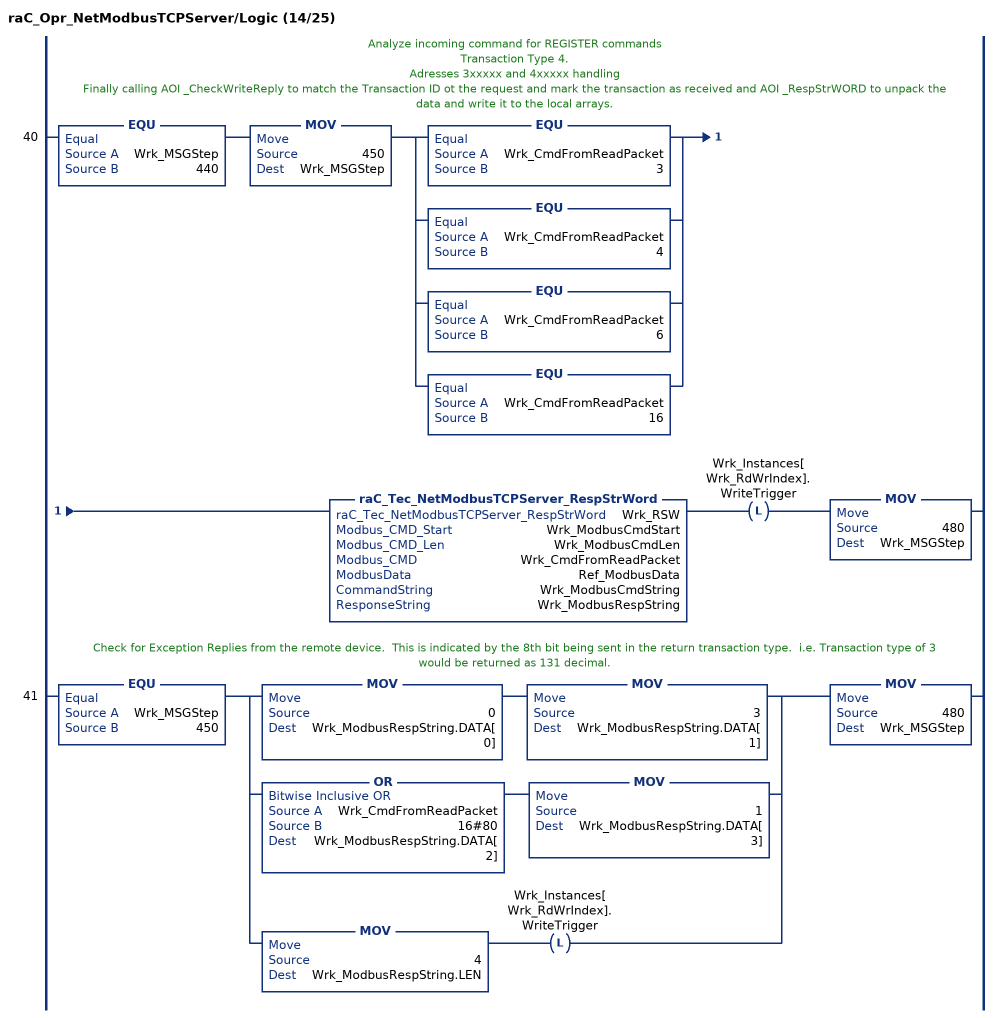
   // Analyze incoming command for REGISTER commands
   // Transaction Type 4.
   // Adresses 3xxxxx and 4xxxxx handling
   // Finally calling AOI _CheckWriteReply to match the Transaction ID ot the request and mark the transaction as received and AOI _RespStrWORD to unpack the data and write it to the local arrays.
   40: EQU(Wrk_MSGStep,440)MOV(450,Wrk_MSGStep)[EQU(Wrk_CmdFromReadPacket,3) ,EQU(Wrk_CmdFromReadPacket,4) ,EQU(Wrk_CmdFromReadPacket,6) ,EQU(Wrk_CmdFromReadPacket,16) ]raC_Tec_NetModbusTCPServer_RespStrWord(Wrk_RSW,Wrk_ModbusCmdStart,Wrk_ModbusCmdLen,Wrk_CmdFromReadPacket,Ref_ModbusData,Wrk_ModbusCmdString,Wrk_ModbusRespString)OTL(Wrk_Instances[Wrk_RdWrIndex].WriteTrigger)MOV(480,Wrk_MSGStep);
   // Check for Exception Replies from the remote device.  This is indicated by the 8th bit being sent in the return transaction type.  i.e. Transaction type of 3 would be returned as 131 decimal.
   41: EQU(Wrk_MSGStep,450)[MOV(0,Wrk_ModbusRespString.DATA[0]) MOV(3,Wrk_ModbusRespString.DATA[1]) ,OR(Wrk_CmdFromReadPacket,16#80,Wrk_ModbusRespString.DATA[2]) MOV(1,Wrk_ModbusRespString.DATA[3]) ,MOV(4,Wrk_ModbusRespString.LEN) OTL(Wrk_Instances[Wrk_RdWrIndex].WriteTrigger) ]MOV(480,Wrk_MSGStep);
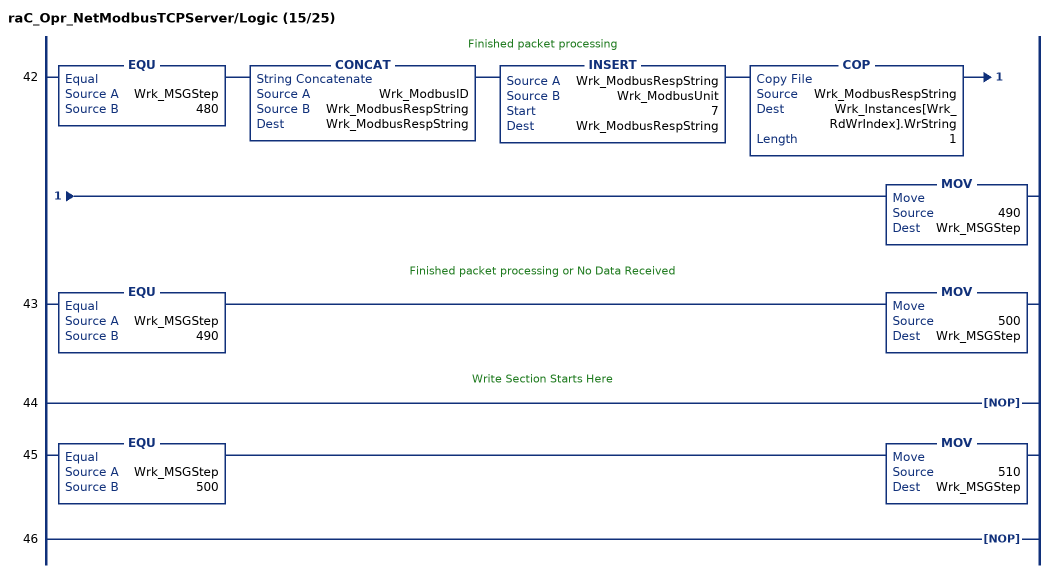
   // Finished packet processing
   42: EQU(Wrk_MSGStep,480)CONCAT(Wrk_ModbusID,Wrk_ModbusRespString,Wrk_ModbusRespString)INSERT(Wrk_ModbusRespString,Wrk_ModbusUnit,7,Wrk_ModbusRespString)COP(Wrk_ModbusRespString,Wrk_Instances[Wrk_RdWrIndex].WrString,1)MOV(490,Wrk_MSGStep);
   // Finished packet processing or No Data Received
   43: EQU(Wrk_MSGStep,490)MOV(500,Wrk_MSGStep);
   // Write Section Starts Here
   44: NOP();
   45: EQU(Wrk_MSGStep,500)MOV(510,Wrk_MSGStep);
   46: NOP();
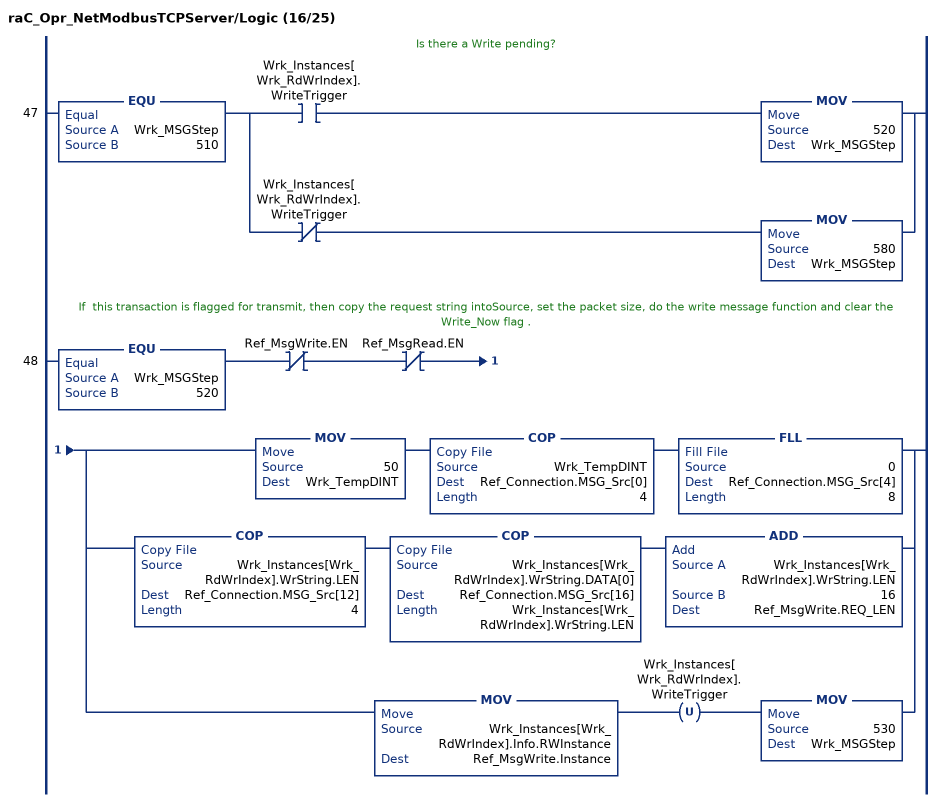
   // Is there a Write pending?
   47: EQU(Wrk_MSGStep,510)[XIC(Wrk_Instances[Wrk_RdWrIndex].WriteTrigger) MOV(520,Wrk_MSGStep) ,XIO(Wrk_Instances[Wrk_RdWrIndex].WriteTrigger) MOV(580,Wrk_MSGStep) ];
   // If  this transaction is flagged for transmit, then copy the request string intoSource, set the packet size, do the write message function and clear the Write_Now flag .
   48: EQU(Wrk_MSGStep,520)XIO(Ref_MsgWrite.EN)XIO(Ref_MsgRead.EN)[MOV(50,Wrk_TempDINT) COP(Wrk_TempDINT,Ref_Connection.MSG_Src[0],4) FLL(0,Ref_Connection.MSG_Src[4],8) ,COP(Wrk_Instances[Wrk_RdWrIndex].WrString.LEN,Ref_Connection.MSG_Src[12],4) COP(Wrk_Instances[Wrk_RdWrIndex].WrString.DATA[0],Ref_Connection.MSG_Src[16],Wrk_Instances[Wrk_RdWrIndex].WrString.LEN) ADD(Wrk_Instances[Wrk_RdWrIndex].WrString.LEN,16,Ref_MsgWrite.REQ_LEN) ,MOV(Wrk_Instances[Wrk_RdWrIndex].Info.RWInstance,Ref_MsgWrite.Instance) OTU(Wrk_Instances[Wrk_RdWrIndex].WriteTrigger) MOV(530,Wrk_MSGStep) ];
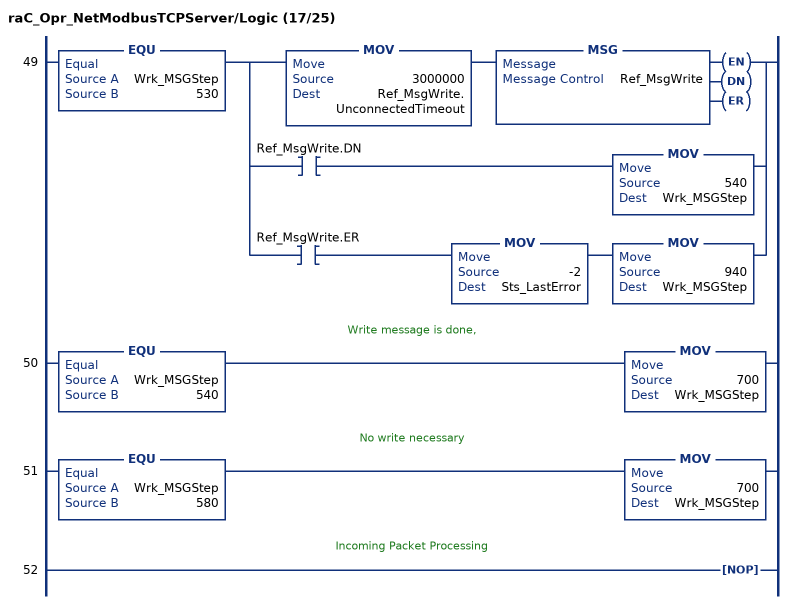
   49: EQU(Wrk_MSGStep,530)[MOV(3000000,Ref_MsgWrite.UnconnectedTimeout) MSG(Ref_MsgWrite) ,XIC(Ref_MsgWrite.DN) MOV(540,Wrk_MSGStep) ,XIC(Ref_MsgWrite.ER) MOV(-2,Sts_LastError) MOV(940,Wrk_MSGStep) ];
   // Write message is done,
   50: EQU(Wrk_MSGStep,540)MOV(700,Wrk_MSGStep);
   // No write necessary
   51: EQU(Wrk_MSGStep,580)MOV(700,Wrk_MSGStep);
   // Incoming Packet Processing
   52: NOP();
